FUNCTION_BLOCK Test_AssertEquals_STRING EXTENDS T_UnitTestBase
VAR
    AssertionUnderTest : T_Assertion;
    STRING_Variable : STRING := 'Cucumber';
END_VAR

// Test the assertion...
AssertionUnderTest.AssertEquals_STRING(
    Expected := 'Radish',
    Actual   := STRING_Variable,
    VariableName := 'STRING_Variable'); 
    
// Assert that the assertion failed...
Assertion.AssertEquals_BOOL(Expected     := TRUE,
                            Actual       := AssertionUnderTest.AssertionFailed,
                            VariableName := 'AssertionUnderTest.AssertionFailed');

// Check the assertion worked...  
CheckAssertion(NextState := 0);

END_FUNCTION_BLOCK

(* stored: Version 1.1.0.1, ProductVersion 3.1.4024.11
   POU Test_AssertEquals_STRING: Id {db994c4a-d987-4378-af34-b707794fadd7}, SpecialFunc None *)
